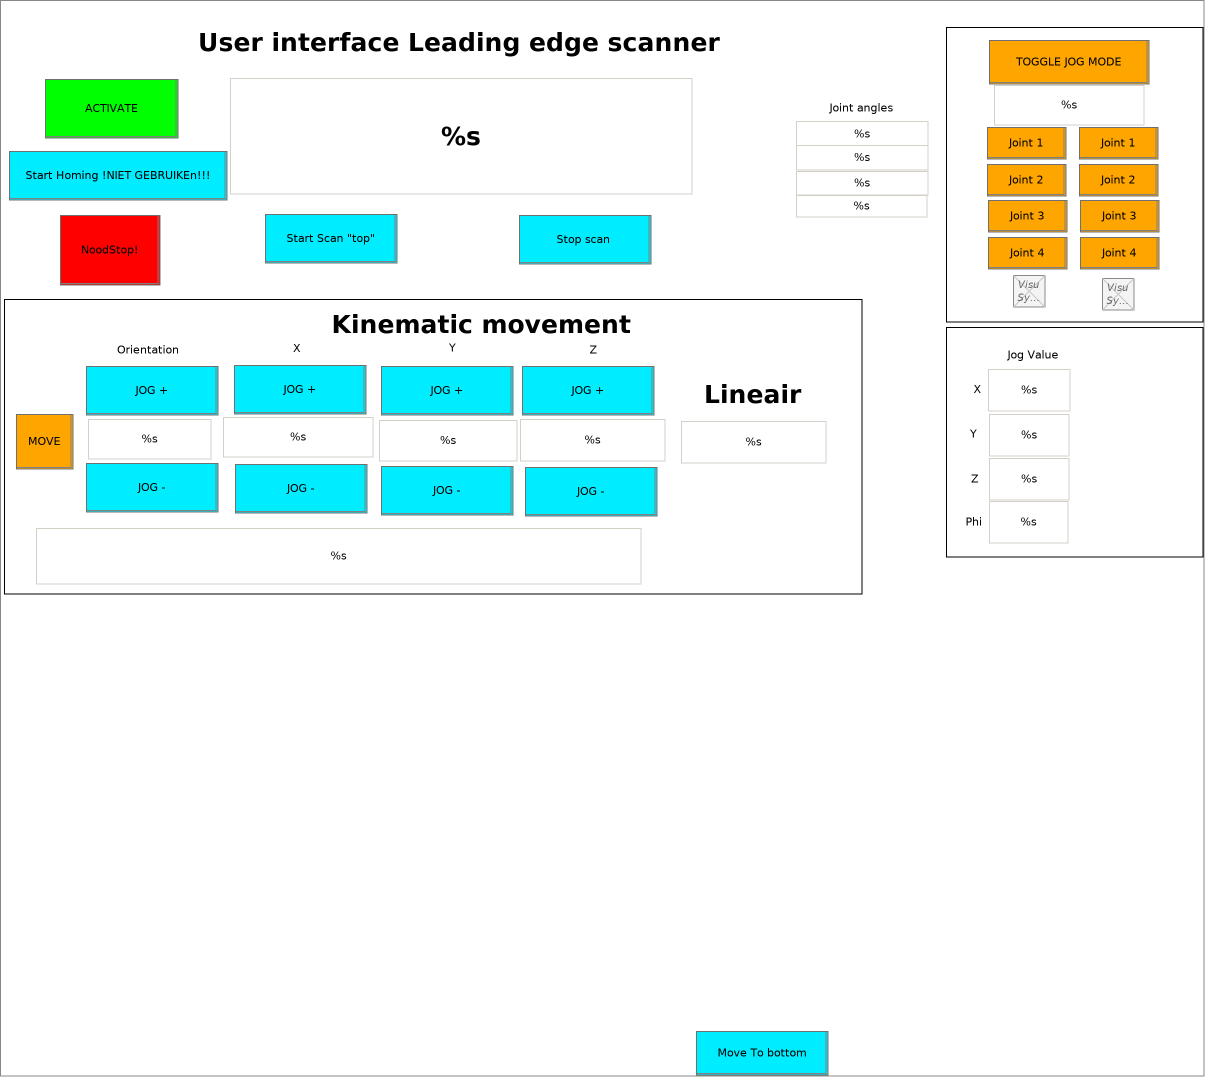
VISUALIZATION Visualization  // 1205x1077
    Rectangle (4,299 858x295)
    Rectangle (946,27 257x295)
    Rectangle (946,327 257x230)
    Textfield (230,78 462x116), "%s", text variable: MAIN.sStateDesc
    Button (9,151 218x49), "Start Homing !NIET GEBRUIKEn!!!"
        tap MAIN.btHoming
    Button (45,79 133x59), "ACTIVATE"
        tap MAIN.btActivator
        OnMouseClick: execute { MAIN.iState:= 5; }
    Button (60,215 100x70), "NoodStop!"
        OnMouseDown: execute { MAIN.iState:= 800; MAIN.sStateDesc := '!ERROR NOODSTOP!'; }
    Button (987,127 79x32), "Joint 1"
        OnMouseDown: execute { MAIN.MotorJog := 1; }
        OnMouseUp: execute { MAIN.MotorJog := 100; }
    Button (989,40 160x44), "TOGGLE JOG MODE"
        toggle MAIN.JOG;
        OnMouseClick: execute { MAIN.iState := 11; }
    Button (1079,127 79x32), "Joint 1"
        OnMouseDown: execute { MAIN.MotorJog := 5; }
        OnMouseUp: execute { MAIN.MotorJog := 100; }
    Button (987,164 79x32), "Joint 2"
        OnMouseDown: execute { MAIN.MotorJog := 2; }
        OnMouseUp: execute { MAIN.MotorJog := 100; }
    Button (1079,164 79x32), "Joint 2"
        OnMouseDown: execute { MAIN.MotorJog := 6; }
        OnMouseUp: execute { MAIN.MotorJog := 100; }
    Button (988,200 79x32), "Joint 3"
        OnMouseDown: execute { MAIN.MotorJog := 3; }
        OnMouseUp: execute { MAIN.MotorJog := 100; }
    Button (1080,200 79x32), "Joint 3"
        OnMouseDown: execute { MAIN.MotorJog := 7; }
        OnMouseUp: execute { MAIN.MotorJog := 100; }
    Button (988,237 79x32), "Joint 4"
        OnMouseDown: execute { MAIN.MotorJog := 4; }
        OnMouseUp: execute { MAIN.MotorJog := 100; }
    Button (1080,237 79x32), "Joint 4"
        OnMouseDown: execute { MAIN.MotorJog := 8; }
        OnMouseUp: execute { MAIN.MotorJog := 100; }
    Textfield (994,85 150x40), "%s", text variable: MAIN.sJogDesk
    Button (16,414 57x55), "MOVE"
        OnMouseClick: execute { MAIN.iState := 12; }
    Textfield (223,417 150x40), "%s", text variable: MAIN.X_coordinate
        OnMouseClick: write MAIN.X_coordinate via InputWithLimits, min -700, max 700, format %
    Image (1102,278 32x32), image: VisuSymbols.Symbols.ArrowCircle2LeftRightLeft
    Image (1013,275 32x32), image: VisuSymbols.Symbols.ArrowCircle2RightRightLeft
    Textfield (379,420 138x41), "%s", text variable: MAIN.Y_coordinate
        OnMouseClick: write MAIN.Y_coordinate via Default, min -700, max 700, format %
    Textfield (520,419 145x42), "%s", text variable: MAIN.Z_coordinate
        OnMouseClick: write MAIN.Z_coordinate via Default, min 0, max 827, format %
    Textfield (796,121 132x26), "%s", text variable: MAIN.CalculatedJ1
    Textfield (796,145 132x25), "%s", text variable: MAIN.CalculatedJ2
    Textfield (796,171 132x24), "%s", text variable: MAIN.CalculatedJ3
    Textfield (796,195 131x22), "%s", text variable: MAIN.CalculatedJ4
    Textfield (88,419 123x40), "%s", text variable: MAIN.Graden_orientatie
        OnMouseClick: write MAIN.Graden_orientatie via InputWithLimits, min -360, max 360, format %
    Label (257,337 80x23), "X"
    Label (398,325 109x46), "Y"
    Label (539,327 109x46), "Z"
    Label (69,327 162x46), "Orientation"
    Button (234,365 132x49), "JOG +"
        OnMouseUp: execute {  }
        OnMouseDown: execute {
            MAIN.X_coordinate := MAIN.X_coordinate + MAIN.JOG_Value_X_axis;
            MAIN.iState := 12;
            //MAIN.iState := 13;
        }
    Button (235,464 132x49), "JOG -"
        OnMouseUp: execute {  }
        OnMouseDown: execute {
            MAIN.X_coordinate := MAIN.X_coordinate - MAIN.JOG_Value_X_axis;
            MAIN.iState := 12;
            //MAIN.iState := 13;
        }
    Button (381,366 132x49), "JOG +"
        OnMouseUp: execute {  }
        OnMouseDown: execute {
            MAIN.Y_coordinate := MAIN.Y_coordinate + MAIN.JOG_Value_Y_axis;
            MAIN.iState := 12;
            //MAIN.iState := 13;
        }
    Button (522,366 132x49), "JOG +"
        OnMouseUp: execute {  }
        OnMouseDown: execute {
            MAIN.Z_coordinate := MAIN.Z_coordinate + MAIN.JOG_Value_Z_axis;
            MAIN.iState := 12;
            //MAIN.iState := 13;
        }
    Button (381,466 132x49), "JOG -"
        OnMouseUp: execute {  }
        OnMouseDown: execute {
            MAIN.Y_coordinate := MAIN.Y_coordinate - MAIN.JOG_Value_Y_axis;
            MAIN.iState := 12;
            //MAIN.iState := 13;
        }
    Button (525,467 132x49), "JOG -"
        OnMouseUp: execute {  }
        OnMouseDown: execute {
            MAIN.Z_coordinate := MAIN.Z_coordinate - MAIN.JOG_Value_Z_axis;
            MAIN.iState := 12;
            //MAIN.iState := 13;
        }
    Button (86,366 132x49), "JOG +"
        OnMouseUp: execute {  }
        OnMouseDown: execute {
            MAIN.Graden_orientatie := MAIN.Graden_orientatie + MAIN.JOG_Value_Phi_axis;
            MAIN.iState := 12;
            //MAIN.iState := 13;
        }
    Button (86,463 132x49), "JOG -"
        OnMouseUp: execute {  }
        OnMouseDown: execute {
            MAIN.Graden_orientatie := MAIN.Graden_orientatie - MAIN.JOG_Value_Phi_axis;
            MAIN.iState := 12;
            //MAIN.iState := 13;
        }
    Textfield (988,369 82x42), "%s", text variable: MAIN.JOG_Value_X_axis
        OnMouseClick: write MAIN.JOG_Value_X_axis via Default, format 10
    Label (952,332 162x46), "Jog Value"
    Label (953,361 49x57), "X"
    Label (931,405 85x58), "Y"
    Label (939,452 72x54), "Z"
    Textfield (989,414 80x42), "%s", text variable: MAIN.JOG_Value_Y_axis
        OnMouseClick: write MAIN.JOG_Value_Y_axis via Default, format 10
    Textfield (989,458 80x42), "%s", text variable: MAIN.JOG_Value_Z_axis
        OnMouseClick: write MAIN.JOG_Value_Z_axis via Default, format 10
    Label (938,495 72x54), "Phi"
    Textfield (989,501 79x42), "%s", text variable: MAIN.JOG_Value_Phi_axis
        OnMouseClick: write MAIN.JOG_Value_Phi_axis via Default, format 10
    Textfield (36,528 605x56), "%s", text variable: MAIN.sNoodstop
    Label (226,301 511x46), "Kinematic movement"
    Label (623,371 260x46), "Lineair"
    Textfield (681,421 145x42), "%s", text variable: MAIN.displacement_mm
        OnMouseClick: write MAIN.displacement_mm via Default, min 0, max 2000000, format %
    Button (265,214 132x49), "Start Scan "top""
        toggle MAIN.PosScan
        OnMouseDown: execute { MAIN.iState := 15; }
        OnMouseClick: execute { MAIN.iState := 15; }
        OnMouseUp: execute {  }
    Button (696,1031 132x44), "Move To bottom"
        toggle MAIN.PosScan
        OnMouseUp: execute {  }
        OnMouseClick: execute { MAIN.iState := 16; }
        OnMouseDown: execute { MAIN.iState := 15; }
    Button (519,215 132x49), "Stop scan"
        toggle MAIN.PosScan
        OnMouseDown: execute { MAIN.iState := 15; }
        OnMouseClick: execute { MAIN.iState := 10; }
        OnMouseUp: execute {  }
    Label (54,19 810x46), "User interface Leading edge scanner"
    Label (794,85 135x46), "Joint angles"
END_VISUALIZATION

(* stored: Version 1.1.0.1, ProductVersion 3.1.4022.18
   Visu Visualization: Id {403ed305-28d1-4c9f-8cdc-f97540241a8d} *)
